PROGRAM Display_Pos
VAR
END_VAR

IF GVL.iiAtPos = 1 THEN
	GVL.qxDIsplay_Pos := 'HOME';
ELSIF GVL.iiAtPos = 2 THEN
	GVL.qxDIsplay_Pos := 'A';
ELSIF GVL.iiAtPos = 3 THEN
	GVL.qxDIsplay_Pos := 'B';
ELSIF GVL.iiAtPos = 4 THEN
	GVL.qxDIsplay_Pos := 'C';
ELSIF GVL.iiAtPos = 5 THEN
	GVL.qxDIsplay_Pos := 'D';
ELSIF GVL.iiAtPos = 6 THEN
	GVL.qxDIsplay_Pos := 'STOP AGV';
END_IF

END_PROGRAM

(* stored: Version 1.1.0.1, ProductVersion 3.1.4024.12
   POU Display_Pos: Id {35d3a6d9-f24d-41c0-b52f-7088e0cdbd49}, SpecialFunc None *)
